Fanuc KAREL source: kb00187.KL

PROGRAM KB00187
%STACKSIZE=65535
%PRIORITY=65535
%NOLOCKGROUP
VAR
P1 : REAL
RESULT : REAL
BEGIN
P1=1.0
-- UNRESOLVED_PC line 8 opcodes [27 22 76 23] marker_code=16
END KB00187
